(* PLC project Generated.project, CODESYS CODESYS V3.5 SP19 Patch 1 *)
(* stored: creationDateTime 2026-09-06T13:00:42.428691, modificationDateTime 2026-09-06T13:00:42.428691 *)

(* ======================================================================= 💾 ST_fbWinchSpeedLearning_Cell — Cellule de vitesse apprise ─────────────────────────────────────────────────────────────── 🎯 Rôle : Cellule unitaire de la table d'apprentissage vitesse par palier 📄 Doc metier : DOC/AF/AF_Partie-10_Fonction_Winch_v2.1.md ======================================================================= *)
TYPE ST_fbWinchSpeedLearning_Cell : STRUCT
  Valid : BOOL;  (* Cellule validee (vitesse apprise exploitable) *)
  SpeedMps : REAL;  (* Vitesse apprise (m/s) *)
  SampleCount : UDINT;  (* Compteur d'echantillons collectes *)
END_STRUCT;
END_TYPE

(* ======================================================================= ⚙️ ST_fbWinchSpeedLearning_Cfg — Enveloppes de plausibilite par palier ─────────────────────────────────────────────────────────────── 🎯 Rôle : Bornes min/max de vitesse apprise par palier + seuil d'echantillons 📄 Doc metier : DOC/AF/AF_Partie-10_Fonction_Winch_v2.1.md ======================================================================= *)
TYPE ST_fbWinchSpeedLearning_Cfg : STRUCT
  MinSpeedMps : ARRAY[1..5] OF REAL;  (* Borne min vitesse apprise par palier (m/s) *)
  MaxSpeedMps : ARRAY[1..5] OF REAL;  (* Borne max vitesse apprise par palier (m/s) *)
  MinSamples : UDINT;  (* Nb min d'echantillons pour valider une cellule *)
END_STRUCT;
END_TYPE

(* ======================================================================= 💾 ST_fbWinchSpeedLearning_Table — Table RETAIN apprentissage vitesse ─────────────────────────────────────────────────────────────── 🎯 Rôle : Matrice {axe x sens x charge/vide x palier} de vitesses apprises 📄 Doc metier : DOC/AF/AF_Partie-10_Fonction_Winch_v2.1.md ======================================================================= *)
TYPE ST_fbWinchSpeedLearning_Table : STRUCT
  Cell : ARRAY[1..2, 1..2, 1..2, 1..5] OF ST_fbWinchSpeedLearning_Cell;  (* [axe][sens][charge][palier] axe : 1=M1, 2=M2 sens : 1=montee, 2=descente charge : 1=vide, 2=charge palier : 1..5 *)
END_STRUCT;
END_TYPE

(* ======================================================================= 💾 FB_WinchSpeedLearning — Collecteur passif vitesse par palier ─────────────────────────────────────────────────────────────── 🎯 Rôle : Apprentissage passif des vitesses reelles par palier (RETAIN) 📄 Doc metier : DOC/AF/AF_Partie-10_Fonction_Winch_v2.1.md 🔒 Collecteur pur : aucune commande moteur, aucune surveillance survitesse ======================================================================= *)
FUNCTION_BLOCK FB_WinchSpeedLearning
  VAR_INPUT
    Enable : BOOL;  (* === CONTRAT LIGHT (Enable) === --> [CMD] Autorisation generale FB (TRUE=Autorise) *)
    LearnStart : BOOL;  (* --> [CMD] Bit IHM lancer apprentissage *)
    WinchId : INT;  (* --> [CMD] Axe cible (1=M1, 2=M2) *)
    ReqAscent : BOOL;  (* --> [HW] Mesure active montée *)
    ReqDescend : BOOL;  (* --> [HW] Mesure active descente *)
    StepNumber : INT;  (* --> [HW] Palier actif (1..5) *)
    MeasuredSpeedMps : REAL;  (* --> [HW] Vitesse mesuree (m/s) *)
    MeasuredSpeedValid : BOOL;  (* --> [HW] Mesure exploitable *)
    LoadPresent : BOOL;  (* --> [HW] Charge presente (TRUE=charge, FALSE=vide) *)
    StableForLearn : BOOL;  (* --> [HW] Conditions stables pour apprentissage *)
    Config : ST_fbWinchSpeedLearning_Cfg;  (* === REGLAGES & CONFIGURATION === --> [CFG] Enveloppes de plausibilite par palier *)
  END_VAR
  VAR_OUTPUT
    Ready : BOOL;  (* === CONTRAT LIGHT (Ready) === <-- [STAT] FB pret (Enable) *)
    Learning : BOOL;  (* === ETATS & DIAGNOSTIC === <-- [STAT] Collecte en cours *)
    TableComplete : BOOL;  (* <-- [STAT] Table charge ET vide complete *)
    LampLearn : BOOL;  (* <-- [STAT] Voyant IHM apprentissage *)
    CellsFilled : INT;  (* <-- [DIAG] Nombre de cellules validees *)
    CellsTotal : INT;  (* <-- [DIAG] Nombre total de cellules *)
  END_VAR
  VAR_IN_OUT
    Table : ST_fbWinchSpeedLearning_Table;  (* === STRUCTURES DE DONNEES PARTAGEES === <-> [BUS] Table RETAIN apprentissage *)
  END_VAR
  VAR
    LearnRequested : BOOL;  (* === VARIABLES LOCALES CALCULEES === . [LOC] Bit IHM + Enable *)
    MeasureUsable : BOOL;  (* . [LOC] Mesure valide + conditions stables *)
    SensActive : BOOL;  (* . [LOC] Un seul sens actif *)
    SensConflict : BOOL;  (* . [LOC] Deux sens actifs : collecte interdite *)
    StepInRange : BOOL;  (* . [LOC] Palier dans 1..5 *)
    AxeInRange : BOOL;  (* . [LOC] Axe dans 1..2 *)
    ContextValid : BOOL;  (* . [LOC] Sens, palier et axe dans le domaine *)
    CollectAllowed : BOOL;  (* . [LOC] Conditions de collecte reunies *)
    SpeedPlausible : BOOL;  (* . [LOC] Vitesse dans l'enveloppe du palier *)
    SensIdx : INT;  (* . [LOC] Index sens (1=montee, 2=descente) *)
    ChargeIdx : INT;  (* . [LOC] Index charge (1=vide, 2=charge) *)
    CurrentCell : ST_fbWinchSpeedLearning_Cell;  (* . [LOC] Cellule courante *)
    AxeIdx : INT;  (* . [LOC] Index axe boucle *)
    SensLoopIdx : INT;  (* . [LOC] Index sens boucle *)
    ChargeLoopIdx : INT;  (* . [LOC] Index charge boucle *)
    PalierIdx : INT;  (* . [LOC] Index palier boucle *)
    CST_AxeCount : INT := 2;  (* Nombre d'axes (M1, M2) *)
    CST_SensCount : INT := 2;  (* Nombre de sens (ascending, descending) *)
    CST_ChargeCount : INT := 2;  (* Nombre d'etats de charge (vide, charge) *)
    CST_PalierCount : INT := 5;  (* Nombre de paliers (1..5) *)
    CST_IdxAscent : INT := 1;  (* Index sens ascending *)
    CST_IdxDescent : INT := 2;  (* Index sens descending *)
    CST_IdxVide : INT := 1;  (* Index charge vide *)
    CST_IdxCharge : INT := 2;  (* Index charge presente *)
  END_VAR

            

{region "§1 Gate et conditions de collecte"}
Ready := Enable;
Learning := FALSE;
LampLearn := FALSE;

// Conditions de collecte scindees (lisibilite Watch, <=3 termes par predicat)
LearnRequested := Enable AND LearnStart;
MeasureUsable := MeasuredSpeedValid AND StableForLearn;
SensConflict := ReqAscent AND ReqDescend;
SensActive := (ReqAscent OR ReqDescend) AND NOT SensConflict;
StepInRange := (StepNumber >= 1) AND (StepNumber <= CST_PalierCount);
AxeInRange := (WinchId >= 1) AND (WinchId <= CST_AxeCount);
ContextValid := SensActive AND StepInRange AND AxeInRange;
CollectAllowed := LearnRequested AND MeasureUsable AND ContextValid;
{endregion}

{region "§2 Collecte passive"}
IF CollectAllowed THEN
    // Index sens et charge
    IF ReqAscent THEN SensIdx := CST_IdxAscent; ELSE SensIdx := CST_IdxDescent; END_IF;
    IF LoadPresent THEN ChargeIdx := CST_IdxCharge; ELSE ChargeIdx := CST_IdxVide; END_IF;

    // Plausibilite : vitesse dans l'enveloppe du palier (borne min/max)
    SpeedPlausible := (MeasuredSpeedMps >= Config.MinSpeedMps[StepNumber])
                      AND (MeasuredSpeedMps <= Config.MaxSpeedMps[StepNumber]);

    CurrentCell := Table.Cell[WinchId, SensIdx, ChargeIdx, StepNumber];
    IF SpeedPlausible THEN
        // Accumulation (moyenne glissante)
        IF CurrentCell.SampleCount = 0 THEN
            CurrentCell.SpeedMps := MeasuredSpeedMps;
            CurrentCell.SampleCount := 1;
        ELSE
            CurrentCell.SpeedMps := (CurrentCell.SpeedMps * UDINT_TO_REAL(CurrentCell.SampleCount) + MeasuredSpeedMps)
                                    / UDINT_TO_REAL(CurrentCell.SampleCount + 1);
            CurrentCell.SampleCount := CurrentCell.SampleCount + 1;
        END_IF;
        CurrentCell.Valid := (CurrentCell.SampleCount >= Config.MinSamples);
    ELSE
        // Valeur hors enveloppe -> cellule invalidee
        CurrentCell.Valid := FALSE;
        CurrentCell.SampleCount := 0;
        CurrentCell.SpeedMps := 0.0;
    END_IF;
    Table.Cell[WinchId, SensIdx, ChargeIdx, StepNumber] := CurrentCell;

    Learning := TRUE;
    LampLearn := TRUE;
END_IF;
{endregion}

{region "§3 Comptage et completude"}
CellsTotal := CST_AxeCount * CST_SensCount * CST_ChargeCount * CST_PalierCount;
CellsFilled := 0;
FOR AxeIdx := 1 TO CST_AxeCount DO
    FOR SensLoopIdx := 1 TO CST_SensCount DO
        FOR ChargeLoopIdx := 1 TO CST_ChargeCount DO
            FOR PalierIdx := 1 TO CST_PalierCount DO
                IF Table.Cell[AxeIdx, SensLoopIdx, ChargeLoopIdx, PalierIdx].Valid THEN
                    CellsFilled := CellsFilled + 1;
                END_IF;
            END_FOR;
        END_FOR;
    END_FOR;
END_FOR;
TableComplete := (CellsFilled >= CellsTotal);
{endregion}

          
END_FUNCTION_BLOCK
